PROGRAM POU_DALI_Sensor_Prog
VAR
	fbDALI102Dimmer1Sensor	 : FB_DALI102Dimmer1Switch(POU_Comm.fbKL6821Communication);
	bInitialize              : BOOL := FALSE;
	motionSensor			 : BOOL;
 	bRecallMaxLevel          : BOOL;
 	bRecallMinLevel          : BOOL;
 	//bOn                      : BOOL;
 	//bOff                     : BOOL;
  	bToggle                  : BOOL;
  	bGoToScene               : BOOL;
  	nScene                   : BYTE;
  	bSetLevel                : BOOL;
  	nLevel                   : BYTE := 254;
  	nLevelMemoryMode         : BYTE := 90;
  	nReferenceDeviceAddress  : BYTE;
  	tCycleActualLevel        : TIME := T#5S;
  	nOptions                 : DWORD := 0;
	nActualLevel             : BYTE;
END_VAR

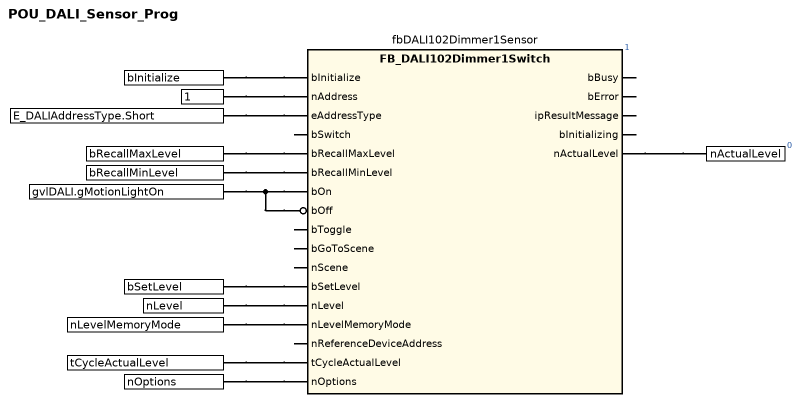
nActualLevel := fbDALI102Dimmer1Sensor.nActualLevel;
fbDALI102Dimmer1Sensor(
    bInitialize := bInitialize,
    nAddress := 1,
    eAddressType := E_DALIAddressType.Short,
    bRecallMaxLevel := bRecallMaxLevel,
    bRecallMinLevel := bRecallMinLevel,
    bOn := gvlDALI.gMotionLightOn,
    bOff := NOT gvlDALI.gMotionLightOn,
    bSetLevel := bSetLevel,
    nLevel := nLevel,
    nLevelMemoryMode := nLevelMemoryMode,
    tCycleActualLevel := tCycleActualLevel,
    nOptions := nOptions); // FB_DALI102Dimmer1Switch

END_PROGRAM

(* stored: Version 1.1.0.1, ProductVersion 3.1.4024.15
   POU POU_DALI_Sensor_Prog: Id {d712b85d-be6d-47a7-bbe2-86a17c83b76c}, SpecialFunc None *)
